FUNCTION_BLOCK FB_System_WDT_Ablaufsteuerung
VAR_IN_OUT
	Zustand						: ST_System_WDT_Zustand;
	Stellwert					: ST_System_WDT_Stellwert;
	Steuerung					: ST_System_WDT_Steuerung;
END_VAR
VAR_INPUT
	Zustand_Stellventil_Netz_WW	: ST_SVs_Zustand;
	Zustand_Stellventil_Netz_KW	: ST_SVs_Zustand;
	Zustand_Stellventil_AFA		: ST_SVs_504_505_Zustand;
	Zustand_Pumpe_Netz			: ST_PU_Zustand;
	Zustand_Pumpe				: ST_PU_Zustand;
	Zustand_Regelventil			: ST_RV_Zustand;
END_VAR
VAR_OUTPUT
END_VAR
VAR
	E_System_WDT_Zustand_Status_Nachl_Stellventil	: SINT;
	E_System_WDT_Zustand_Status_Nachl_Pumpe			: SINT;
	E_System_WDT_Zustand_Status_Betrieb				: SINT;
	E_System_WDT_Zustand_Status_Betrieb_Sperre		: SINT;
	E_System_WDT_Zustand_Status_Vorl_Pumpe			: SINT;
	E_System_WDT_Zustand_Status_Vorl_Stellventil	: SINT;
	E_System_WDT_Zustand_Status_Betriebsbereit		: SINT;
	E_System_WDT_Zustand_Status_Stoerung			: SINT;
	E_System_WDT_Zustand_Status_Idle_Sperre			: SINT;
END_VAR

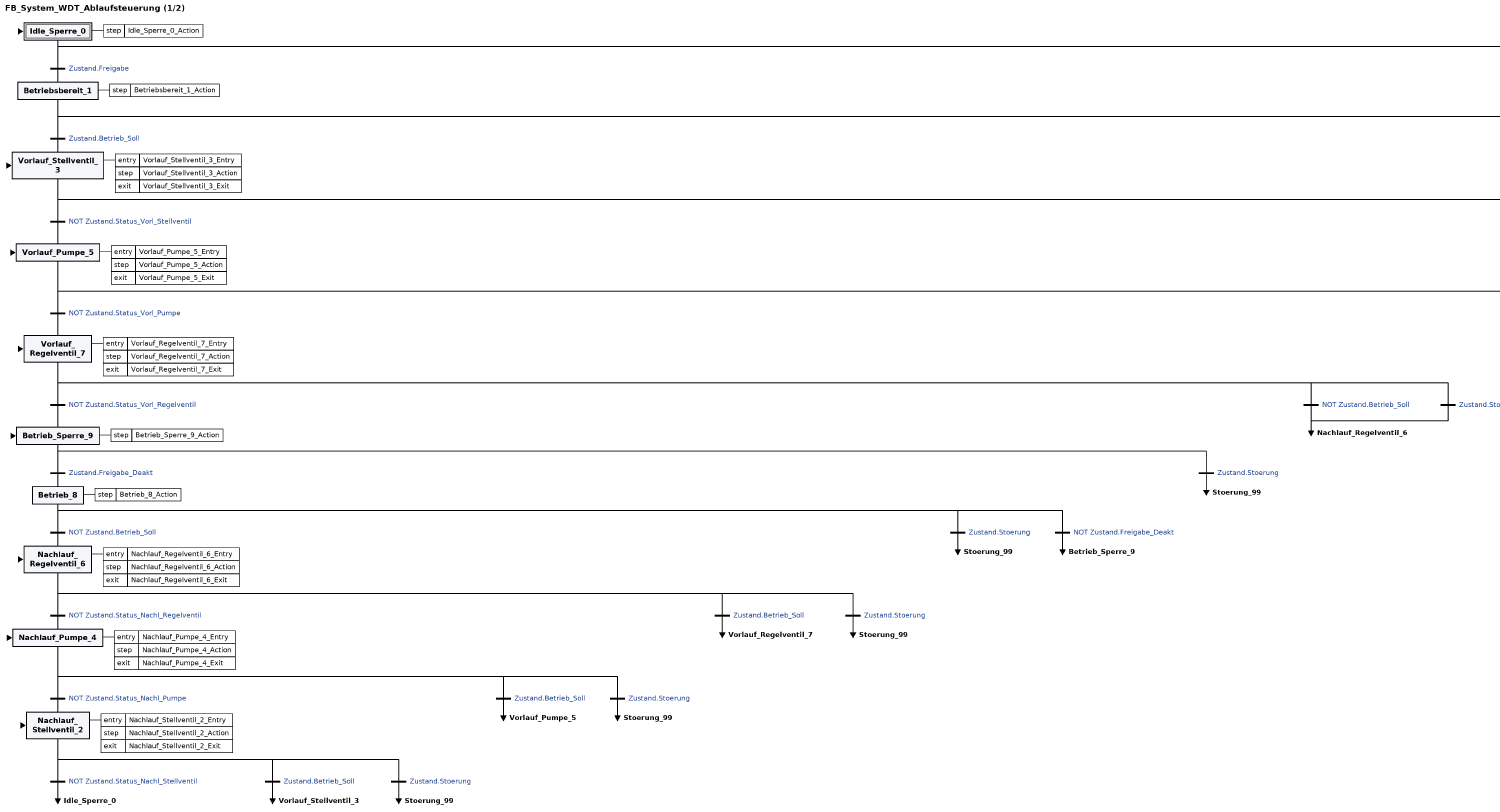
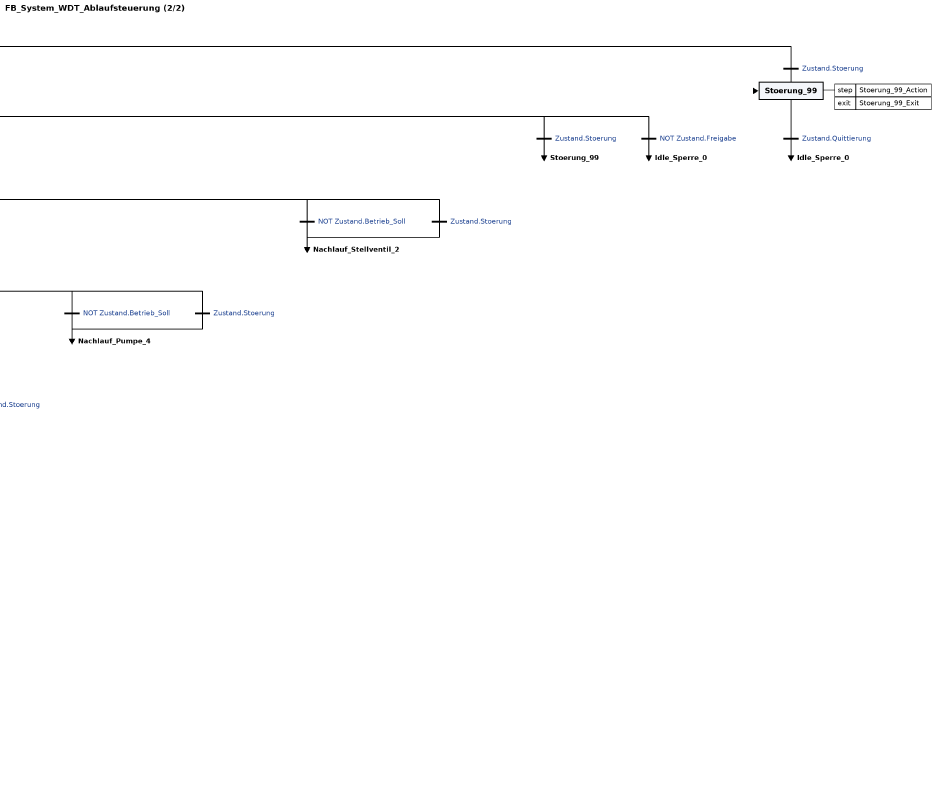
INITIAL_STEP Idle_Sperre_0:
    Idle_Sperre_0_Action(N);  // step action
END_STEP
TRANSITION FROM Idle_Sperre_0 TO Betriebsbereit_1
    := Zustand.Freigabe;
END_TRANSITION
TRANSITION FROM Idle_Sperre_0 TO Stoerung_99
    := Zustand.Stoerung;
END_TRANSITION
STEP Stoerung_99:
    Stoerung_99_Action(N);  // step action
    Stoerung_99_Exit(P0);  // exit action
END_STEP
TRANSITION FROM Stoerung_99 TO Idle_Sperre_0
    := Zustand.Quittierung;
END_TRANSITION
STEP Betriebsbereit_1:
    Betriebsbereit_1_Action(N);  // step action
END_STEP
TRANSITION FROM Betriebsbereit_1 TO Vorlauf_Stellventil_3
    := Zustand.Betrieb_Soll;
END_TRANSITION
TRANSITION FROM Betriebsbereit_1 TO Stoerung_99
    := Zustand.Stoerung;
END_TRANSITION
TRANSITION FROM Betriebsbereit_1 TO Idle_Sperre_0
    := NOT Zustand.Freigabe;
END_TRANSITION
STEP Vorlauf_Stellventil_3:
    Vorlauf_Stellventil_3_Entry(P1);  // entry action
    Vorlauf_Stellventil_3_Action(N);  // step action
    Vorlauf_Stellventil_3_Exit(P0);  // exit action
END_STEP
TRANSITION FROM Vorlauf_Stellventil_3 TO Vorlauf_Pumpe_5
    := NOT Zustand.Status_Vorl_Stellventil;
END_TRANSITION
TRANSITION FROM Vorlauf_Stellventil_3 TO Nachlauf_Stellventil_2
    := NOT Zustand.Betrieb_Soll;
END_TRANSITION
TRANSITION FROM Vorlauf_Stellventil_3 TO Nachlauf_Stellventil_2
    := Zustand.Stoerung;
END_TRANSITION
STEP Vorlauf_Pumpe_5:
    Vorlauf_Pumpe_5_Entry(P1);  // entry action
    Vorlauf_Pumpe_5_Action(N);  // step action
    Vorlauf_Pumpe_5_Exit(P0);  // exit action
END_STEP
TRANSITION FROM Vorlauf_Pumpe_5 TO Vorlauf_Regelventil_7
    := NOT Zustand.Status_Vorl_Pumpe;
END_TRANSITION
TRANSITION FROM Vorlauf_Pumpe_5 TO Nachlauf_Pumpe_4
    := NOT Zustand.Betrieb_Soll;
END_TRANSITION
TRANSITION FROM Vorlauf_Pumpe_5 TO Nachlauf_Pumpe_4
    := Zustand.Stoerung;
END_TRANSITION
STEP Vorlauf_Regelventil_7:
    Vorlauf_Regelventil_7_Entry(P1);  // entry action
    Vorlauf_Regelventil_7_Action(N);  // step action
    Vorlauf_Regelventil_7_Exit(P0);  // exit action
END_STEP
TRANSITION FROM Vorlauf_Regelventil_7 TO Betrieb_Sperre_9
    := NOT Zustand.Status_Vorl_Regelventil;
END_TRANSITION
TRANSITION FROM Vorlauf_Regelventil_7 TO Nachlauf_Regelventil_6
    := NOT Zustand.Betrieb_Soll;
END_TRANSITION
TRANSITION FROM Vorlauf_Regelventil_7 TO Nachlauf_Regelventil_6
    := Zustand.Stoerung;
END_TRANSITION
STEP Betrieb_Sperre_9:
    Betrieb_Sperre_9_Action(N);  // step action
END_STEP
TRANSITION FROM Betrieb_Sperre_9 TO Betrieb_8
    := Zustand.Freigabe_Deakt;
END_TRANSITION
TRANSITION FROM Betrieb_Sperre_9 TO Stoerung_99
    := Zustand.Stoerung;
END_TRANSITION
STEP Betrieb_8:
    Betrieb_8_Action(N);  // step action
END_STEP
TRANSITION FROM Betrieb_8 TO Nachlauf_Regelventil_6
    := NOT Zustand.Betrieb_Soll;
END_TRANSITION
TRANSITION FROM Betrieb_8 TO Stoerung_99
    := Zustand.Stoerung;
END_TRANSITION
TRANSITION FROM Betrieb_8 TO Betrieb_Sperre_9
    := NOT Zustand.Freigabe_Deakt;
END_TRANSITION
STEP Nachlauf_Regelventil_6:
    Nachlauf_Regelventil_6_Entry(P1);  // entry action
    Nachlauf_Regelventil_6_Action(N);  // step action
    Nachlauf_Regelventil_6_Exit(P0);  // exit action
END_STEP
TRANSITION FROM Nachlauf_Regelventil_6 TO Nachlauf_Pumpe_4
    := NOT Zustand.Status_Nachl_Regelventil;
END_TRANSITION
TRANSITION FROM Nachlauf_Regelventil_6 TO Vorlauf_Regelventil_7
    := Zustand.Betrieb_Soll;
END_TRANSITION
TRANSITION FROM Nachlauf_Regelventil_6 TO Stoerung_99
    := Zustand.Stoerung;
END_TRANSITION
STEP Nachlauf_Pumpe_4:
    Nachlauf_Pumpe_4_Entry(P1);  // entry action
    Nachlauf_Pumpe_4_Action(N);  // step action
    Nachlauf_Pumpe_4_Exit(P0);  // exit action
END_STEP
TRANSITION FROM Nachlauf_Pumpe_4 TO Nachlauf_Stellventil_2
    := NOT Zustand.Status_Nachl_Pumpe;
END_TRANSITION
TRANSITION FROM Nachlauf_Pumpe_4 TO Vorlauf_Pumpe_5
    := Zustand.Betrieb_Soll;
END_TRANSITION
TRANSITION FROM Nachlauf_Pumpe_4 TO Stoerung_99
    := Zustand.Stoerung;
END_TRANSITION
STEP Nachlauf_Stellventil_2:
    Nachlauf_Stellventil_2_Entry(P1);  // entry action
    Nachlauf_Stellventil_2_Action(N);  // step action
    Nachlauf_Stellventil_2_Exit(P0);  // exit action
END_STEP
TRANSITION FROM Nachlauf_Stellventil_2 TO Idle_Sperre_0
    := NOT Zustand.Status_Nachl_Stellventil;
END_TRANSITION
TRANSITION FROM Nachlauf_Stellventil_2 TO Vorlauf_Stellventil_3
    := Zustand.Betrieb_Soll;
END_TRANSITION
TRANSITION FROM Nachlauf_Stellventil_2 TO Stoerung_99
    := Zustand.Stoerung;
END_TRANSITION

ACTION Betrieb_8_Action:
(* Stellwert setzen *)
Stellwert.Anford_Stellventil_Netz	:= TRUE;
Stellwert.Anford_Pumpe_Netz	:= TRUE;
Stellwert.Anford_Stellventil		:= TRUE;
Stellwert.Anford_Pumpe		:= TRUE;
Stellwert.Anford_Regelventil		:= TRUE;

(* Zustand setzen *)
Zustand.Betrieb				:= TRUE;
Zustand.Status				:= E_System_WDT_Zustand_Status_Betrieb;
END_ACTION

ACTION Betrieb_Sperre_9_Action:
(* Stellwert setzen *)
Stellwert.Anford_Stellventil_Netz	:= TRUE;
Stellwert.Anford_Pumpe_Netz	:= TRUE;
Stellwert.Anford_Stellventil		:= TRUE;
Stellwert.Anford_Pumpe		:= TRUE;
Stellwert.Anford_Regelventil		:= TRUE;

(* Zustand setzen *)
Zustand.Betrieb				:= TRUE;
Zustand.Status				:= E_System_WDT_Zustand_Status_Betrieb_Sperre;
END_ACTION

ACTION Betriebsbereit_1_Action:
(* Stellwert setzen *)
Stellwert.Anford_Stellventil_Netz	:= FALSE;
Stellwert.Anford_Pumpe_Netz	:= FALSE;
Stellwert.Anford_Stellventil		:= FALSE;
Stellwert.Anford_Pumpe		:= FALSE;
Stellwert.Anford_Regelventil		:= FALSE;
Stellwert.Anford_Aussenfassadenaktivierung	:= FALSE;

(* Zustand setzen *)
Zustand.Betrieb			:= FALSE;
Zustand.Status			:= E_System_WDT_Zustand_Status_Betriebsbereit;
END_ACTION

ACTION Idle_Sperre_0_Action:
(* Stellwert setzen *)
Stellwert.Anford_Stellventil_Netz	:= FALSE;
Stellwert.Anford_Pumpe_Netz	:= FALSE;
Stellwert.Anford_Stellventil		:= FALSE;
Stellwert.Anford_Pumpe		:= FALSE;
Stellwert.Anford_Regelventil		:= FALSE;
Stellwert.Anford_Aussenfassadenaktivierung	:= FALSE;

(* Zustand setzen *)
Zustand.Betrieb			:= FALSE;
Zustand.Status			:= E_System_WDT_Zustand_Status_Idle_Sperre;

(* Quittierungszustand auf False setzen, damit das System bei einer erneuten Störung nicht direkt wieder angeschaltet wird *)
Steuerung.Quittierung	:= FALSE;
END_ACTION

ACTION Nachlauf_Pumpe_4_Action:
(* Stellwert setzen *)
Stellwert.Anford_Stellventil_Netz	:= TRUE;
Stellwert.Anford_Pumpe_Netz	:= FALSE;
Stellwert.Anford_Stellventil		:= TRUE;
Stellwert.Anford_Pumpe		:= FALSE;
Stellwert.Anford_Regelventil		:= FALSE;
Stellwert.Anford_Aussenfassadenaktivierung	:= FALSE;


(* Zustand setzen *)
Zustand.Betrieb				:= FALSE;
Zustand.Status				:= E_System_WDT_Zustand_Status_Nachl_Pumpe;
Zustand.Status_Nachl_Pumpe	:= Zustand_Pumpe.Betrieb OR Zustand_Pumpe.Status_Nachl OR (Zustand.Modus_viaNetz AND(Zustand_Pumpe_Netz.Betrieb OR Zustand_Pumpe_Netz.Status_Nachl));
END_ACTION

ACTION Nachlauf_Pumpe_4_Entry:
Zustand.Status_Nachl_Pumpe	:= TRUE;
END_ACTION

ACTION Nachlauf_Pumpe_4_Exit:
Zustand.Status_Nachl_Pumpe	:= FALSE;
END_ACTION

ACTION Nachlauf_Regelventil_6_Action:
(* Stellwert setzen *)
Stellwert.Anford_Stellventil_Netz	:= TRUE;
Stellwert.Anford_Pumpe_Netz	:= TRUE;
Stellwert.Anford_Stellventil		:= TRUE;
Stellwert.Anford_Pumpe		:= TRUE;
Stellwert.Anford_Regelventil		:= FALSE;
Stellwert.Anford_Aussenfassadenaktivierung	:= FALSE;


(* Zustand setzen *)
Zustand.Betrieb					:= FALSE;
Zustand.Status					:= E_System_WDT_Zustand_Status_Nachl_Regelventil;
Zustand.Status_Nachl_Regelventil	:= Zustand_Regelventil.Betrieb OR Zustand_Regelventil.Status_Nachl;
END_ACTION

ACTION Nachlauf_Regelventil_6_Entry:
Zustand.Status_Nachl_Regelventil		:= TRUE;
END_ACTION

ACTION Nachlauf_Regelventil_6_Exit:
Zustand.Status_Nachl_Regelventil		:= FALSE;
END_ACTION

ACTION Nachlauf_Stellventil_2_Action:
(* Stellwert setzen *)
Stellwert.Anford_Stellventil_Netz	:= FALSE;
Stellwert.Anford_Pumpe_Netz	:= FALSE;
Stellwert.Anford_Stellventil		:= FALSE;
Stellwert.Anford_Pumpe		:= FALSE;
Stellwert.Anford_Regelventil		:= FALSE;
Stellwert.Anford_Aussenfassadenaktivierung	:= FALSE;


(* Zustand setzen *)
Zustand.Betrieb				:= FALSE;
Zustand.Status				:= E_System_WDT_Zustand_Status_Nachl_Stellventil;
Zustand.Status_Nachl_Stellventil :=
Zustand.Modus_viaNetz AND (
	Zustand.Modus_Heizung AND (
		Zustand_Stellventil_Netz_WW.Stellung OR Zustand_Stellventil_Netz_WW.Stellungwechsel10
	)
	OR (
		Zustand.Modus_Kuehlung AND (
			Zustand_Stellventil_Netz_KW.Stellung OR Zustand_Stellventil_Netz_KW.Stellungwechsel10
		)
	)
);
END_ACTION

ACTION Nachlauf_Stellventil_2_Entry:
Zustand.Status_Nachl_Stellventil	:= TRUE;
END_ACTION

ACTION Nachlauf_Stellventil_2_Exit:
Zustand.Status_Nachl_Stellventil	:= FALSE;
END_ACTION

ACTION Stoerung_99_Action:
(* Stellwert setzen *)
Stellwert.Anford_Stellventil_Netz	:= FALSE;
Stellwert.Anford_Pumpe_Netz	:= FALSE;
Stellwert.Anford_Stellventil		:= FALSE;
Stellwert.Anford_Pumpe		:= FALSE;
Stellwert.Anford_Regelventil		:= FALSE;
Stellwert.Anford_Aussenfassadenaktivierung	:= FALSE;

(* Zustand setzen *)
Zustand.Betrieb			:= FALSE;
Zustand.Stoerung			:= TRUE;
Zustand.Status			:= E_System_WDT_Zustand_Status_Stoerung;
END_ACTION

ACTION Stoerung_99_Exit:
Zustand.Stoerung	:= FALSE;
END_ACTION

ACTION Vorlauf_Pumpe_5_Action:
(* Stellwert setzen *)
Stellwert.Anford_Stellventil_Netz	:= TRUE;
Stellwert.Anford_Pumpe_Netz	:= TRUE;
Stellwert.Anford_Stellventil		:= TRUE;
Stellwert.Anford_Pumpe		:= TRUE;
Stellwert.Anford_Regelventil		:= FALSE;
Stellwert.Anford_Aussenfassadenaktivierung	:= FALSE;


(* Zustand setzen *)
Zustand.Betrieb				:= FALSE;
Zustand.Status				:= E_System_WDT_Zustand_Status_Vorl_Pumpe;
Zustand.Status_Vorl_Pumpe	:=
NOT(
	Zustand_Pumpe.Betrieb AND NOT Zustand_Pumpe.Status_Vorl
)
OR
(
	Zustand.Modus_viaNetz AND NOT(
		Zustand_Pumpe_Netz.Betrieb AND NOT Zustand_Pumpe_Netz.Status_Vorl
	)
)
;
END_ACTION

ACTION Vorlauf_Pumpe_5_Entry:
Zustand.Status_Vorl_Pumpe	:= TRUE;
END_ACTION

ACTION Vorlauf_Pumpe_5_Exit:
Zustand.Status_Vorl_Pumpe	:= FALSE;
END_ACTION

ACTION Vorlauf_Regelventil_7_Action:
(* Stellwert setzen *)
Stellwert.Anford_Stellventil_Netz	:= TRUE;
Stellwert.Anford_Pumpe_Netz	:= TRUE;
Stellwert.Anford_Stellventil		:= TRUE;
Stellwert.Anford_Pumpe		:= TRUE;
Stellwert.Anford_Regelventil		:= TRUE;


(* Zustand setzen *)
Zustand.Betrieb				:= FALSE;
Zustand.Status				:= E_System_WDT_Zustand_Status_Vorl_Regelventil;
Zustand.Status_Vorl_Regelventil	:= NOT(Zustand_Regelventil.Betrieb AND NOT Zustand_Regelventil.Status_Vorl);
END_ACTION

ACTION Vorlauf_Regelventil_7_Entry:
Zustand.Status_Vorl_Regelventil	:= TRUE;
END_ACTION

ACTION Vorlauf_Regelventil_7_Exit:
Zustand.Status_Vorl_Regelventil		:= FALSE;
END_ACTION

ACTION Vorlauf_Stellventil_3_Action:
(* Stellwert setzen *)
Stellwert.Anford_Stellventil_Netz	:= TRUE;
Stellwert.Anford_Pumpe_Netz	:= FALSE;
Stellwert.Anford_Stellventil		:= TRUE;
Stellwert.Anford_Pumpe		:= FALSE;
Stellwert.Anford_Regelventil		:= FALSE;
Stellwert.Anford_Aussenfassadenaktivierung	:= FALSE;


(* Zustand setzen *)
Zustand.Betrieb				:= FALSE;
Zustand.Status				:= E_System_WDT_Zustand_Status_Vorl_Stellventil;
Zustand.Status_Vorl_Stellventil	:=
(
	Zustand.Modus_viaNetz AND
	(
		(
		Zustand.Modus_Heizung AND NOT Zustand_Stellventil_Netz_WW.Stellung AND Zustand_Stellventil_Netz_WW.Stellungwechsel01
		)
		OR
		(
		Zustand.Modus_Kuehlung AND NOT Zustand_Stellventil_Netz_KW.Stellung AND Zustand_Stellventil_Netz_KW.Stellungwechsel01
		)
	)
)
OR
(
	Zustand.Modus_viaAussenfassade AND NOT Zustand_Stellventil_AFA.Stellungrueckmeldung1_505
);
END_ACTION

ACTION Vorlauf_Stellventil_3_Entry:
Zustand.Status_Vorl_Stellventil	:= TRUE;
END_ACTION

ACTION Vorlauf_Stellventil_3_Exit:
Zustand.Status_Vorl_Stellventil	:= FALSE;
END_ACTION

END_FUNCTION_BLOCK

(* stored: Version 1.1.0.1, ProductVersion 3.1.4024.9
   POU FB_System_WDT_Ablaufsteuerung: Id {899e0ef7-93b5-4b1c-8eeb-1007876fe6f1}, SpecialFunc None
   Action Betrieb_8_Action: Id {3eb0ec85-441f-4d07-9555-c773c4773f60}
   Action Betrieb_Sperre_9_Action: Id {81acfcff-ee81-465e-b289-dbfdee8acc8d}
   Action Betriebsbereit_1_Action: Id {cb883fa3-7e14-41de-bf36-b6f1ad572761}
   Action Idle_Sperre_0_Action: Id {5b07653e-a429-473a-bf1c-6a9aca2bc86d}
   Action Nachlauf_Pumpe_4_Action: Id {5a9be1fb-e3c7-49c5-8a3a-0c5de450ac59}
   Action Nachlauf_Pumpe_4_Entry: Id {d4efe7db-cbd7-4921-af6d-91fd60e8047d}
   Action Nachlauf_Pumpe_4_Exit: Id {ea4a6e65-fc2c-47b1-a88e-7c8e2b718159}
   Action Nachlauf_Regelventil_6_Action: Id {98bcbd22-3d31-4a8e-a615-710573b477a5}
   Action Nachlauf_Regelventil_6_Entry: Id {7c266614-8c64-4495-ad17-7ef0b123a9c4}
   Action Nachlauf_Regelventil_6_Exit: Id {1214f0a8-b03f-4931-a872-67901a7519fb}
   Action Nachlauf_Stellventil_2_Action: Id {fd31c1c1-290f-4dec-970c-8e2578470e48}
   Action Nachlauf_Stellventil_2_Entry: Id {25763129-3e8c-4288-a373-999cbe9c4772}
   Action Nachlauf_Stellventil_2_Exit: Id {dd677da1-ef49-479a-bf00-be0cba550a0c}
   Action Stoerung_99_Action: Id {5d0b2f04-d734-46d6-8323-3fcbfa937bd4}
   Action Stoerung_99_Exit: Id {9c6b46f9-9356-432e-b62a-73629a8824d5}
   Action Vorlauf_Pumpe_5_Action: Id {ac55b952-3260-4f1f-8530-1e8ebf187c42}
   Action Vorlauf_Pumpe_5_Entry: Id {b1893d7d-7bca-43b3-a65a-8ccab83fc8d7}
   Action Vorlauf_Pumpe_5_Exit: Id {0f4504f3-4d9f-4bcd-b193-74283f99934a}
   Action Vorlauf_Regelventil_7_Action: Id {e68c7193-da43-4353-b10d-9ef60549c5d5}
   Action Vorlauf_Regelventil_7_Entry: Id {08c9e90f-b979-4c70-89e1-ba1e1af31dd9}
   Action Vorlauf_Regelventil_7_Exit: Id {e6c394b9-fd71-4734-b616-abc6a42837b3}
   Action Vorlauf_Stellventil_3_Action: Id {aa99ae5b-40a1-4d68-82cb-1fb0e0980676}
   Action Vorlauf_Stellventil_3_Entry: Id {a602fa8a-e61c-4a49-ab40-dc2cf5ca13a4}
   Action Vorlauf_Stellventil_3_Exit: Id {8eaf671d-7e90-4b36-a26e-3020f005aea5} *)
